{attribute 'no_explicit_call' := 'do not call this FB directly'}{attribute 'enable_dynamic_creation'}
FUNCTION_BLOCK FINAL PlaygroundNode EXTENDS Node
VAR
	value1 : _INT(0);
	value2 : _INT(-100);
	value3 : _INT(123);
	minimum : _INT(-10);
	maximum : _INT(20);
	onlyOdd : _BOOL(TRUE);
END_VAR

METHOD PUBLIC Clone : I_Node
VAR
	pNode : POINTER TO PlaygroundNode;
END_VAR
pNode := __NEW(PlaygroundNode);
Clone := pNode^;
END_METHOD

METHOD FB_init : BOOL
VAR_INPUT
	bInitRetains : BOOL; // if TRUE, the retain variables are initialized (warm start / cold start)
	bInCopyCode : BOOL;  // if TRUE, the instance afterwards gets moved into the copy code (online change)
END_VAR
AddParameter('value1', value1)
	.AddMetadata('maximumValue',maximum)
	.AddMetadata('minimumValue',minimum);
AddParameter('value2', value2)
	.AddMetadata('minimumValue',minimum)
	.AddMetadata('onlyOdd', onlyOdd);
	
AddParameter('value3', value3);
END_METHOD

METHOD PROTECTED OnExecute : HRESULT
VAR
END_VAR
END_METHOD

END_FUNCTION_BLOCK

(* stored: Version 1.1.0.1, ProductVersion 3.1.4024.12
   POU PlaygroundNode: Id {8ca5c23c-4555-02eb-0a5c-be06b622d8bb}, SpecialFunc None
   Folder Constructor: Id {2c10e50b-90b9-07c1-37d9-e36ffda387fb}
   Method Clone: Id {700c4e05-dabe-05c6-308a-89726582f81c}
   Method FB_init: Id {0a9418ce-6e4a-0c8c-37e4-3b458b778c8d}
   Method OnExecute: Id {88f02288-f470-0eef-2d40-14e43c04a4a0} *)
